{attribute 'linkalways'} 
{attribute 'no_explicit_call' := 'This FB is a CLASS and must be accessed using methods or properties'}
{attribute 'enable_dynamic_creation'}
FUNCTION_BLOCK GearOutCommand EXTENDS DefaultAsyncCommand
VAR
	axis_ref : REFERENCE TO Tc2_Mc2.Axis_Ref;
	fb : Tc2_Mc2.Mc_GearOut;
END_VAR

METHOD PUBLIC CyclicCall
SUPER^.CyclicCall();
fb(Slave := axis_ref);
END_METHOD

(*FB_Init is always available implicitly and it is used primarily for initialization.
The return value is not evaluated. For a specific influence, you can also declare the
methods explicitly and provide additional code there with the standard initialization
code. You can evaluate the return value.*)
METHOD FB_Init : BOOL
VAR_INPUT
	(* TRUE: the retain variables are initialized (reset warm / reset cold)*)
	bInitRetains : BOOL;
	(* TRUE: the instance will be copied to the copy code afterward (online change)*)
	bInCopyCode	: BOOL;
	axis : REFERENCE TO Mc2Axis;
END_VAR
axis_ref REF= axis.Mc2AxisRef;
END_METHOD

METHOD PROTECTED OnExecuting
VAR_INPUT
	state_control : AsyncCommandStateControl;
END_VAR
fb.Execute := TRUE;

IF fb.Done THEN
	state_control.Next();
	fb.Execute := FALSE;
END_IF

IF fb.Error THEN
	state_control.Error(fb.ErrorId);
	fb.Execute := FALSE;
END_IF
END_METHOD

END_FUNCTION_BLOCK

(* stored: Version 1.1.0.1, ProductVersion 3.1.4026.13
   POU GearOutCommand: Id {566486cd-883b-4947-bfc6-8aa6918e25fb}, SpecialFunc None
   Method CyclicCall: Id {1a5cafdd-9624-4feb-9861-cdeb7f44a12a}
   Method FB_Init: Id {c0ebecbd-f539-4bfc-af6d-1545a3f3758c}
   Method OnExecuting: Id {909b21f5-4617-4270-8661-99246477b699} *)
